RoboDK station: Sheet B.rdk

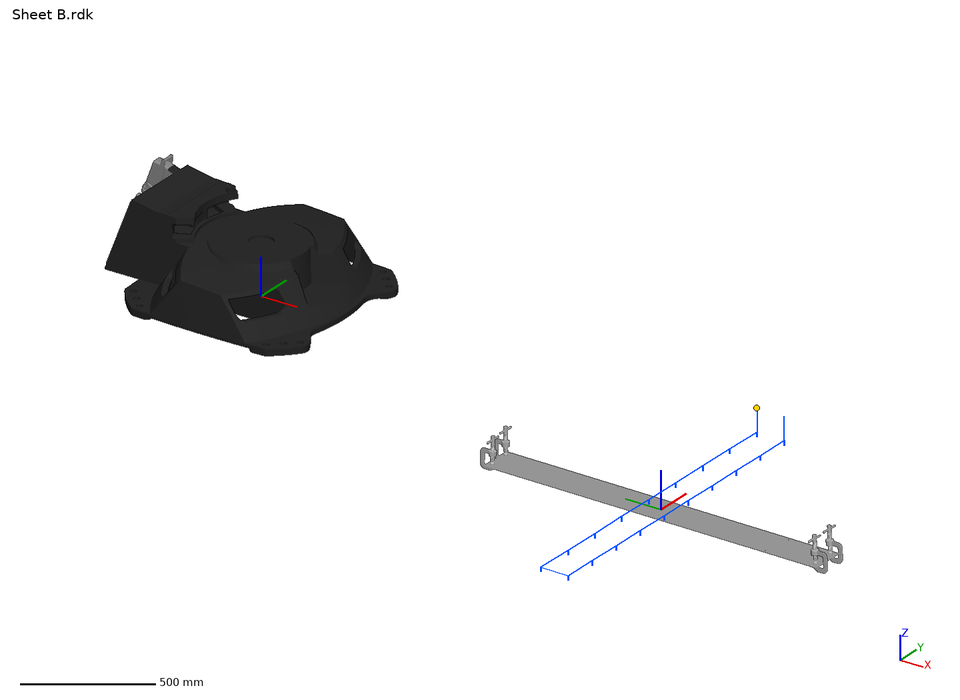
[picture v0: the station drawn from its stored meshes, robots at their saved joint values, targets as dots, program paths as lines]
Station Sheet B (saved by RoboDK 5.2.3). Poses are relative to the parent item; angles as X-Y-Z fixed-axis rotations.
  - frame KUKA KR 210 R2700 extra Base at (0, 0, 0) mm
    - robot KUKA KR 210 R2700 extra: 6 axes, payload 210 kg, reach 2696 mm, repeatability 0.06 mm, weight 1068 kg
        joint limits [-185, -140, -120, -350, -125, -350] to [185, -5, 155, 350, 125, 350]; home [0, -90, 90, 0, 0, 0]; saved at [-4.299, -27.561, 142.534, -183.011, 63.926, -182.019]
      - tool Spindle, TCP at (32, 0, 260) mm, rotated rx 0 ry 39 rz 0 deg, size 157.3 x 72 x 259.9 mm
  - frame Frame 2 at (1800, 0, -372.68) mm, rotated rx 0 ry 0 rz 90 deg
    - object Sheet B-box 2 Hole positioning at (0, 0, 0) mm, rotated rx 0 ry 0 rz 90 deg, 19 curves, geometry from Point 19
    - object Box 2 - Sheet B at (0, 0, 0) mm, size 148.8 x 1500 x 0.8 mm, geometry from Box 2 - Sheet B.stl
  - machining project Point settings: rotZ(0) | rotX(0)*rotY(0) | rotz(0) | onStart | onPathStart | onApproach | onPoint | onRetract | onFinish | SetRPM(%1) | SetTool(%1) | Extruder(%1) | default | default | OutOnMov(%1) | OutOffMov(%1) | onPathFinish | M_RunCode(%1)
  - program Point (106 instructions, listed below)
  - object FinalClamp at (2523.4, 49.78, -312.91) mm, rotated rx 108.73 ry 87.57 rz 18.21 deg, size 145.3 x 71.1 x 72 mm, geometry from FinalClamp.stp
  - object FinalClamp2 at (2526.12, -49.6, -312.39) mm, rotated rx 91.75 ry 86.92 rz 0 deg, size 145.3 x 71.1 x 72 mm, geometry from FinalClamp.stp
  - object FinalClamp3 at (1071.67, 39.98, -310.44) mm, rotated rx -90.18 ry 89.27 rz 0 deg, size 145.3 x 71.1 x 72 mm, geometry from FinalClamp.stp
  - object FinalClamp4 at (1076.14, -50.25, -311.72) mm, rotated rx 89.78 ry 88.55 rz 180 deg, size 145.3 x 71.1 x 72 mm, geometry from FinalClamp.stp
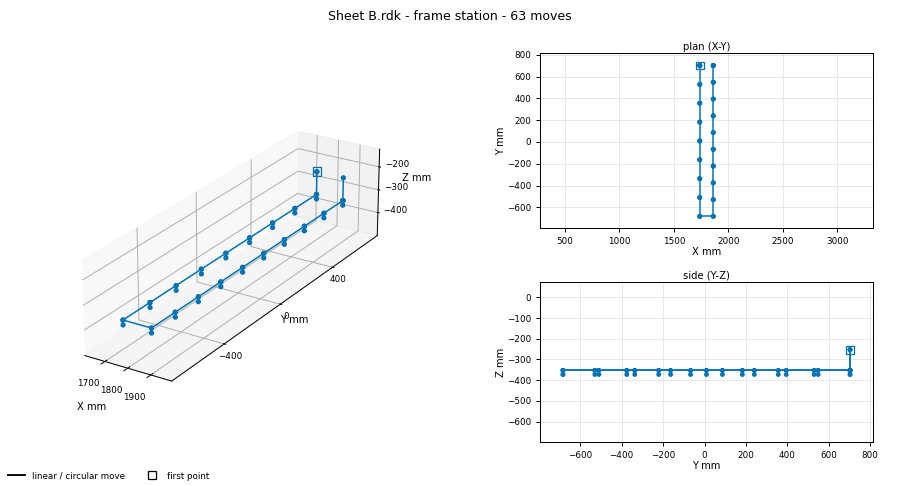
[picture p0: tool path of Sheet B.rdk in frame station, 63 of 63 moves have a stored position in this frame; points joined in program order, loops and branches not executed]

--- program Point (robot KUKA KR 210 R2700 extra) ---
  Smooth(1)
  Set speed (1000.0 mm/s)
  Set Ref.: Frame 2
  Set Tool: Spindle
  Show Spindle
  MoveJ 1 to (702.57, 61.9, 120) mm, rotated rx 180 ry 0 rz 0 deg; joints [4.299, -27.561, 142.534, -176.989, 63.926, -177.981]
  MoveL 2 to (702.57, 61.9, 120) mm, rotated rx 180 ry 0 rz 0 deg; joints [4.299, -27.561, 142.534, -176.989, 63.926, -177.981]
  MoveL 3 to (702.57, 61.9, 20) mm, rotated rx -180 ry 0 rz 0 deg; joints [4.299, -20.368, 138.524, -177.064, 67.105, -177.799]
  MoveL 4 to (702.57, 61.9, 20) mm, rotated rx -180 ry 0 rz 0 deg; joints [4.299, -20.368, 138.524, -177.064, 67.105, -177.799]
  Set speed (50.0 mm/s)
  MoveL 5 to (702.57, 61.9, 0) mm, rotated rx 180 ry 0 rz 0 deg; joints [4.299, -19.028, 137.686, -177.075, 67.605, -177.771]
  MoveL 6 to (702.57, 61.9, 20) mm, rotated rx -180 ry 0 rz 0 deg; joints [4.299, -20.368, 138.524, -177.064, 67.105, -177.799]
  Set speed (1000.0 mm/s)
  MoveL 7 to (529.32, 61.9, 20) mm, rotated rx 180 ry 0 rz 0 deg; joints [3.554, -25.652, 132.554, -177.299, 55.878, -178.753]
  Set speed (50.0 mm/s)
  MoveL 8 to (529.32, 61.9, 0) mm, rotated rx 180 ry 0 rz 0 deg; joints [3.554, -24.341, 131.805, -177.317, 56.439, -178.721]
  MoveL 9 to (529.32, 61.9, 20) mm, rotated rx 180 ry 0 rz 0 deg; joints [3.554, -25.652, 132.554, -177.299, 55.878, -178.753]
  Set speed (1000.0 mm/s)
  MoveL 10 to (356.07, 61.9, 20) mm, rotated rx -180 ry 0 rz 0 deg; joints [3.029, -28.412, 125.559, -177.357, 46.138, -179.478]
  Set speed (50.0 mm/s)
  MoveL 11 to (356.07, 61.9, 0) mm, rotated rx -180 ry 0 rz 0 deg; joints [3.029, -27.178, 124.883, -177.381, 46.696, -179.442]
  MoveL 12 to (356.07, 61.9, 20) mm, rotated rx -180 ry 0 rz 0 deg; joints [3.029, -28.412, 125.559, -177.357, 46.138, -179.478]
  Set speed (1000.0 mm/s)
  MoveL 13 to (182.82, 61.9, 20) mm, rotated rx -180 ry 0 rz 0 deg; joints [2.639, -29.27, 117.725, -177.269, 37.456, -180.117]
  Set speed (50.0 mm/s)
  MoveL 14 to (182.82, 61.9, 0) mm, rotated rx 180 ry 0 rz 0 deg; joints [2.639, -28.127, 117.108, -177.302, 37.982, -180.076]
  MoveL 15 to (182.82, 61.9, 20) mm, rotated rx -180 ry 0 rz 0 deg; joints [2.639, -29.27, 117.725, -177.269, 37.456, -180.117]
  Set speed (1000.0 mm/s)
  MoveL 16 to (9.57, 61.9, 20) mm, rotated rx -180 ry 0 rz 0 deg; joints [2.338, -28.673, 109.123, -177.008, 29.46, -180.788]
  Set speed (50.0 mm/s)
  MoveL 17 to (9.57, 61.9, 0) mm, rotated rx 180 ry 0 rz 0 deg; joints [2.338, -27.615, 108.547, -177.052, 29.941, -180.738]
  MoveL 18 to (9.57, 61.9, 20) mm, rotated rx -180 ry 0 rz 0 deg; joints [2.338, -28.673, 109.123, -177.008, 29.46, -180.788]
  Set speed (1000.0 mm/s)
  MoveL 19 to (-163.68, 61.9, 20) mm, rotated rx 180 ry 0 rz 0 deg; joints [2.098, -26.895, 99.722, -176.45, 21.846, -181.665]
  Set speed (50.0 mm/s)
  MoveL 20 to (-163.68, 61.9, 0) mm, rotated rx -180 ry 0 rz 0 deg; joints [2.098, -25.913, 99.173, -176.516, 22.278, -181.594]
  MoveL 21 to (-163.68, 61.9, 20) mm, rotated rx 180 ry 0 rz 0 deg; joints [2.098, -26.895, 99.722, -176.45, 21.846, -181.665]
  Set speed (1000.0 mm/s)
  MoveL 22 to (-336.93, 61.9, 20) mm, rotated rx -180 ry 0 rz 0 deg; joints [1.903, -24.072, 89.386, -175.162, 14.348, -183.208]
  Set speed (50.0 mm/s)
  MoveL 23 to (-336.93, 61.9, 0) mm, rotated rx -180 ry 0 rz 0 deg; joints [1.903, -23.151, 88.848, -175.285, 14.729, -183.082]
  MoveL 24 to (-336.93, 61.9, 20) mm, rotated rx -180 ry 0 rz 0 deg; joints [1.903, -24.072, 89.386, -175.162, 14.348, -183.208]
  Set speed (1000.0 mm/s)
  MoveL 25 to (-510.18, 61.9, 20) mm, rotated rx -180 ry 0 rz 0 deg; joints [1.741, -20.2, 77.832, -170.578, 6.709, -188.005]
  Set speed (50.0 mm/s)
  MoveL 26 to (-510.18, 61.9, 0) mm, rotated rx -180 ry 0 rz 0 deg; joints [1.741, -19.325, 77.285, -171.014, 7.033, -187.566]
  MoveL 27 to (-510.18, 61.9, 20) mm, rotated rx -180 ry 0 rz 0 deg; joints [1.741, -20.2, 77.832, -170.578, 6.709, -188.005]
  Set speed (1000.0 mm/s)
  MoveL 28 to (-683.43, 61.9, 20) mm, rotated rx -180 ry 0 rz -20 deg; joints [-0.819, -14.541, 63.132, -288.04, 13.606, -87.937]
  Set speed (50.0 mm/s)
  MoveL 29 to (-683.43, 61.9, 0) mm, rotated rx -180 ry 0 rz -20 deg; joints [-0.819, -13.689, 62.537, -287.023, 13.528, -88.983]
  MoveL 30 to (-683.43, 61.9, 20) mm, rotated rx -180 ry 0 rz -20 deg; joints [-0.819, -14.541, 63.132, -288.04, 13.606, -87.937]
  Set speed (1000.0 mm/s)
  MoveL 31 to (-683.43, -61.9, 20) mm, rotated rx 180 ry 0 rz -20 deg; joints [-4, -14.358, 62.684, -288.833, 15.691, -89.578]
  Set speed (50.0 mm/s)
  MoveL 32 to (-683.43, -61.9, 0) mm, rotated rx -180 ry 0 rz -20 deg; joints [-4, -13.506, 62.087, -287.969, 15.61, -90.475]
  MoveL 33 to (-683.43, -61.9, 20) mm, rotated rx 180 ry 0 rz -20 deg; joints [-4, -14.358, 62.684, -288.833, 15.691, -89.578]
  Set speed (1000.0 mm/s)
  MoveL 34 to (-529.43, -61.9, 20) mm, rotated rx 180 ry 0 rz 0 deg; joints [-1.725, -19.7, 76.453, -190.727, 5.842, -170.668]
  Set speed (50.0 mm/s)
  MoveL 35 to (-529.43, -61.9, 0) mm, rotated rx -180 ry 0 rz 0 deg; joints [-1.725, -18.828, 75.903, -190.172, 6.158, -171.226]
  MoveL 36 to (-529.43, -61.9, 20) mm, rotated rx -180 ry 0 rz 0 deg; joints [-1.725, -19.7, 76.453, -190.727, 5.842, -170.668]
  Set speed (1000.0 mm/s)
  MoveL 37 to (-375.43, -61.9, 20) mm, rotated rx -180 ry 0 rz 0 deg; joints [-1.865, -23.305, 86.938, -185.356, 12.672, -176.223]
  Set speed (50.0 mm/s)
  MoveL 38 to (-375.43, -61.9, 0) mm, rotated rx 180 ry 0 rz 0 deg; joints [-1.865, -22.396, 86.4, -185.207, 13.041, -176.376]
  MoveL 39 to (-375.43, -61.9, 20) mm, rotated rx -180 ry 0 rz 0 deg; joints [-1.865, -23.305, 86.938, -185.356, 12.672, -176.223]
  Set speed (1000.0 mm/s)
  MoveL 40 to (-221.43, -61.9, 20) mm, rotated rx -180 ry 0 rz 0 deg; joints [-2.029, -26.067, 96.391, -183.856, 19.346, -177.938]
  Set speed (50.0 mm/s)
  MoveL 41 to (-221.43, -61.9, 0) mm, rotated rx -180 ry 0 rz 0 deg; joints [-2.029, -25.107, 95.847, -183.778, 19.762, -178.021]
  MoveL 42 to (-221.43, -61.9, 20) mm, rotated rx -180 ry 0 rz 0 deg; joints [-2.029, -26.067, 96.391, -183.856, 19.346, -177.938]
  Set speed (1000.0 mm/s)
  MoveL 43 to (-67.43, -61.9, 20) mm, rotated rx -180 ry 0 rz 0 deg; joints [-2.225, -28.017, 105.049, -183.189, 26.045, -178.863]
  Set speed (50.0 mm/s)
  MoveL 44 to (-67.43, -61.9, 0) mm, rotated rx 180 ry 0 rz 0 deg; joints [-2.225, -26.995, 104.487, -183.138, 26.505, -178.921]
  MoveL 45 to (-67.43, -61.9, 20) mm, rotated rx -180 ry 0 rz 0 deg; joints [-2.225, -28.017, 105.049, -183.189, 26.045, -178.863]
  Set speed (1000.0 mm/s)
  MoveL 46 to (86.57, -61.9, 20) mm, rotated rx -180 ry 0 rz 0 deg; joints [-2.462, -29.097, 113.041, -182.849, 32.95, -179.522]
  Set speed (50.0 mm/s)
  MoveL 47 to (86.57, -61.9, 0) mm, rotated rx -180 ry 0 rz 0 deg; joints [-2.462, -28.002, 112.448, -182.812, 33.452, -179.568]
  MoveL 48 to (86.57, -61.9, 20) mm, rotated rx -180 ry 0 rz 0 deg; joints [-2.462, -29.097, 113.041, -182.849, 32.95, -179.522]
  Set speed (1000.0 mm/s)
  MoveL 49 to (240.57, -61.9, 20) mm, rotated rx 180 ry 0 rz 0 deg; joints [-2.757, -29.164, 120.423, -182.685, 40.257, -180.094]
  Set speed (50.0 mm/s)
  MoveL 50 to (240.57, -61.9, 0) mm, rotated rx -180 ry 0 rz 0 deg; joints [-2.757, -27.991, 119.788, -182.656, 40.795, -180.132]
  MoveL 51 to (240.57, -61.9, 20) mm, rotated rx 180 ry 0 rz 0 deg; joints [-2.757, -29.164, 120.423, -182.685, 40.257, -180.094]
  Set speed (1000.0 mm/s)
  MoveL 52 to (394.57, -61.9, 20) mm, rotated rx 180 ry 0 rz 0 deg; joints [-3.132, -27.982, 127.19, -182.643, 48.196, -180.672]
  Set speed (50.0 mm/s)
  MoveL 53 to (394.57, -61.9, 0) mm, rotated rx -180 ry 0 rz 0 deg; joints [-3.132, -26.729, 126.5, -182.621, 48.759, -180.706]
  MoveL 54 to (394.57, -61.9, 20) mm, rotated rx 180 ry 0 rz 0 deg; joints [-3.132, -27.982, 127.19, -182.643, 48.196, -180.672]
  Set speed (1000.0 mm/s)
  MoveL 55 to (548.57, -61.9, 20) mm, rotated rx 180 ry 0 rz 0 deg; joints [-3.624, -25.203, 133.273, -182.717, 57.044, -181.339]
  Set speed (50.0 mm/s)
  MoveL 56 to (548.57, -61.9, 0) mm, rotated rx 180 ry 0 rz 0 deg; joints [-3.624, -23.885, 132.514, -182.7, 57.602, -181.37]
  MoveL 57 to (548.57, -61.9, 20) mm, rotated rx 180 ry 0 rz 0 deg; joints [-3.624, -25.203, 133.273, -182.717, 57.044, -181.339]
  Set speed (1000.0 mm/s)
  MoveL 58 to (702.57, -61.9, 20) mm, rotated rx 180 ry 0 rz 0 deg; joints [-4.299, -20.368, 138.524, -182.936, 67.105, -182.201]
  Set speed (50.0 mm/s)
  MoveL 59 to (702.57, -61.9, 0) mm, rotated rx -180 ry 0 rz 0 deg; joints [-4.299, -19.028, 137.686, -182.925, 67.605, -182.229]
  MoveL 60 to (702.57, -61.9, 20) mm, rotated rx 180 ry 0 rz 0 deg; joints [-4.299, -20.368, 138.524, -182.936, 67.105, -182.201]
  MoveL 61 to (702.57, -61.9, 20) mm, rotated rx 180 ry 0 rz 0 deg; joints [-4.299, -20.368, 138.524, -182.936, 67.105, -182.201]
  Set speed (1000.0 mm/s)
  MoveL 62 to (702.57, -61.9, 20) mm, rotated rx 180 ry 0 rz 0 deg; joints [-4.299, -20.368, 138.524, -182.936, 67.105, -182.201]
  MoveL 63 to (702.57, -61.9, 120) mm, rotated rx -180 ry 0 rz 0 deg; joints [-4.299, -27.561, 142.534, -183.011, 63.926, -182.019]
